// TIA Portal V21 export
TYPE "Std_StrutturaRicetta_SterilizzatoreTubo"
   STRUCT
      NomeFormato : String[20];
      Abilitazione_PompaPistoni : Bool;
      Setpoint_PompaMono : Real;
      Setpoint_PompaPistoni : Real;
      Setpoint_Raffreddatore : Real;
      Setpoint_Sterilizzazione : Real;
   END_STRUCT;
END_TYPE
